(*
A `Execute` method of FB implmenting this interface will be called every control loop cycle.
*)
INTERFACE I_Execute EXTENDS I_Debug

(*
If registered, this method will be executed cyclically.
*)
METHOD Execute
VAR_INPUT
	nPhase: INT;
END_VAR
END_METHOD

END_INTERFACE

(* stored: Version 1.1.0.1
   Itf I_Execute: Id {15413885-918e-40a7-85ba-cc0538727b10}
   Method Execute: Id {d0c1bfc6-1219-4d9b-889c-5e29307fe94f} *)
